// Given a tag value, determines the field number (the upper 29 bits).
FUNCTION F_GetTagFieldNumber : UDINT
VAR_INPUT
    nTag    : UDINT;
END_VAR
VAR
END_VAR


F_GetTagFieldNumber := SHR(nTag, GCL_WireFormat.cTagTypeBits);

END_FUNCTION

(* stored: Version 1.1.0.1
   POU F_GetTagFieldNumber: Id {14c3d22c-3842-4869-a162-a36f91207a6a}, SpecialFunc None *)
